(* Schneider Machine Expert - Basic project Tank_Level_Ultrasonic, file version 3.0.0.0 *)
(* ProjectInformations: Name=Tank_Level_Ultrasonic *)

HARDWARE
  Cpu 0: TM221CE16T
  ModuleExtensionObject 0: TM3AI4/G
  EthernetConfiguration: NetworkName=M221, IpAllocationMode=ByDhcp, IpAddress=192.168.1.10, SubnetMask=255.255.255.0
  SerialLineConfiguration: Baud=Baud19200, Parity=ParityEven, DataBits=DataBits8, StopBits=StopBits1, PhysicalMedium=PhysicalMediumRs485, TransmissionMode=TransmissionModeModbusRtu, SlaveId=1, Addressing=SlaveAddressing
  MastTask: UsePeriodScanMode=false, PeriodScan=100
  FastTask: Period=255
  CpuBehavior: StartingMode=StartAsPreviousState, AutoSaveRamOnEeprom=true, WatchdogPeriod=250

SYMBOLS  (address, symbol, comment, settings)
  %M0       PUMP_RUN  "Pump Running State"
  %M1       LEVEL_LOW  "Level below 1000mm - Start pump"
  %M2       LEVEL_HIGH  "Level above 1500mm - Stop pump"
  %M3       AUTO_CMD  "Auto mode pump command (hysteresis)"
  %M4       SENSOR_VALID  "Sensor reading valid (above dead band)"
  %M5       SENSOR_FAULT  "Sensor fault (below dead band)"
  %S0       SB_COLDSTART  "Indicates or executes a cold start (data initialized to default values)"
  %S1       SB_WARMSTART  "Indicates there was a warm start with data backup"
  %MW0      LVL_RAW  "Raw analog input value (0-10000)"
  %MW1      LVL_DISTANCE  "Distance from sensor in mm (300-5000)"
  %MW2      LVL_ACTUAL  "Actual tank level in mm (0-2000) for HMI"
  %MW10     SP_LOW  "Low level setpoint (1000mm)"
  %MW11     SP_HIGH  "High level setpoint (1500mm)"
  %I0.0     PB_START
  %I0.1     PB_STOP
  %I0.2     ESTOP
  %I0.3     SS_AUTO
  %Q0.0     PUMP_OUT
  %Q0.1     LT_RUN
  %Q0.2     LT_AUTO
  %Q0.3     LT_LOW
  %Q0.4     LT_HIGH
  %IW1.0    LVL_AIN  [Type=Type_4_20mA, Scope=Scope_Customized, Minimum=0, Maximum=10000]

POU Tank_Level_Ultrasonic
  (* SectionNumber=1 *)

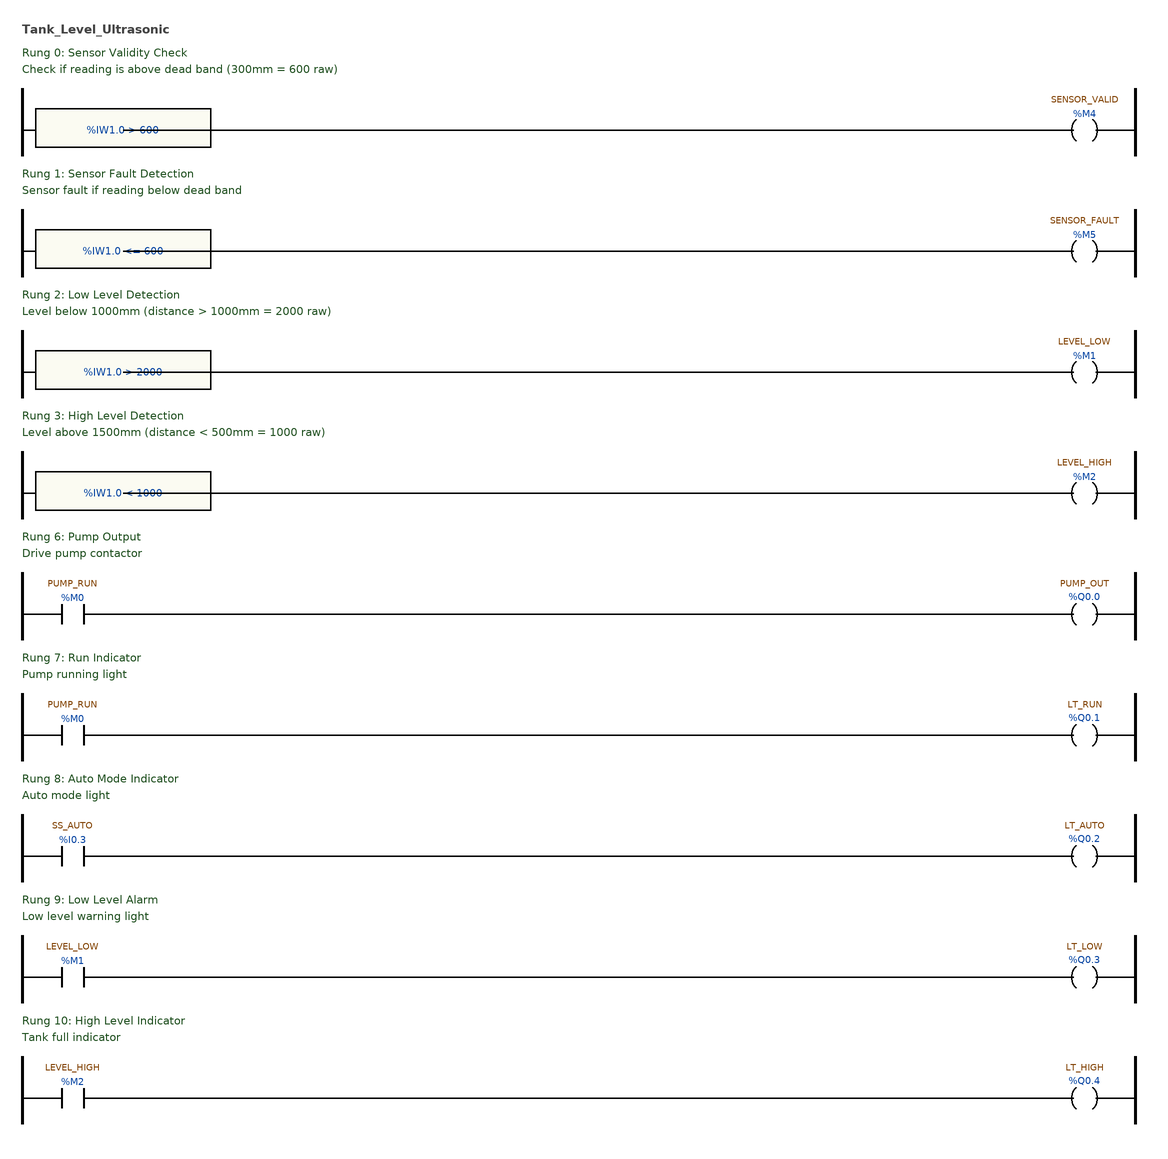

// Rung 0: Sensor Validity Check
// Check if reading is above dead band (300mm = 600 raw)
  LD [ %IW1.0 > 600 ]     (* LVL_AIN *)
  ST %M4                  (* SENSOR_VALID *)
  // as ST:
  //   SENSOR_VALID := LVL_AIN > 600;

// Rung 1: Sensor Fault Detection
// Sensor fault if reading below dead band
  LD [ %IW1.0 <= 600 ]    (* LVL_AIN *)
  ST %M5                  (* SENSOR_FAULT *)
  // as ST:
  //   SENSOR_FAULT := LVL_AIN <= 600;

// Rung 2: Low Level Detection
// Level below 1000mm (distance > 1000mm = 2000 raw)
  LD [ %IW1.0 > 2000 ]    (* LVL_AIN *)
  ST %M1                  (* LEVEL_LOW *)
  // as ST:
  //   LEVEL_LOW := LVL_AIN > 2000;

// Rung 3: High Level Detection
// Level above 1500mm (distance < 500mm = 1000 raw)
  LD [ %IW1.0 < 1000 ]    (* LVL_AIN *)
  ST %M2                  (* LEVEL_HIGH *)
  // as ST:
  //   LEVEL_HIGH := LVL_AIN < 1000;

// Rung 4: Auto Mode Hysteresis
// Start pump at low level, stop at high level (hysteresis 1000-1500mm)
  LD %M1                  (* LEVEL_LOW *)
  OR %M3                  (* AUTO_CMD *)
  ANDN %M2                (* LEVEL_HIGH *)
  AND %M4                 (* SENSOR_VALID *)
  ST %M3                  (* AUTO_CMD *)
  // as ST:
  //   AUTO_CMD := (LEVEL_LOW OR AUTO_CMD) AND NOT LEVEL_HIGH AND SENSOR_VALID;
  (* the ladder stored for this rung does not match its IL; not drawn *)

// Rung 5: Pump Run Control
// Pump runs in Auto mode with AUTO_CMD, or Manual with PB_START
  LD %I0.3                (* SS_AUTO *)
  AND %M3                 (* AUTO_CMD *)
  OR( %I0.0               (* PB_START *)
  OR %M0                  (* PUMP_RUN *)
  ANDN %I0.3              (* SS_AUTO *)
  )
  ANDN %I0.1              (* PB_STOP *)
  ANDN %I0.2              (* ESTOP *)
  AND %M4                 (* SENSOR_VALID *)
  ST %M0                  (* PUMP_RUN *)
  // as ST:
  //   PUMP_RUN := (SS_AUTO AND AUTO_CMD OR (PB_START OR PUMP_RUN) AND NOT SS_AUTO) AND NOT PB_STOP AND NOT ESTOP AND SENSOR_VALID;
  (* the ladder stored for this rung does not match its IL; not drawn *)

// Rung 6: Pump Output
// Drive pump contactor
  LD %M0                  (* PUMP_RUN *)
  ST %Q0.0                (* PUMP_OUT *)
  // as ST:
  //   PUMP_OUT := PUMP_RUN;

// Rung 7: Run Indicator
// Pump running light
  LD %M0                  (* PUMP_RUN *)
  ST %Q0.1                (* LT_RUN *)
  // as ST:
  //   LT_RUN := PUMP_RUN;

// Rung 8: Auto Mode Indicator
// Auto mode light
  LD %I0.3                (* SS_AUTO *)
  ST %Q0.2                (* LT_AUTO *)
  // as ST:
  //   LT_AUTO := SS_AUTO;

// Rung 9: Low Level Alarm
// Low level warning light
  LD %M1                  (* LEVEL_LOW *)
  ST %Q0.3                (* LT_LOW *)
  // as ST:
  //   LT_LOW := LEVEL_LOW;

// Rung 10: High Level Indicator
// Tank full indicator
  LD %M2                  (* LEVEL_HIGH *)
  ST %Q0.4                (* LT_HIGH *)
  // as ST:
  //   LT_HIGH := LEVEL_HIGH;

// Rung 11: HMI Raw Level
// Copy raw analog value to %MW0 for HMI access
  LD %S1                  (* SB_WARMSTART *)
  OR %S0                  (* SB_COLDSTART *)
  [%MW0 := %IW1.0]        (* LVL_RAW, LVL_AIN *)
  // as ST:
  //   IF SB_WARMSTART OR SB_COLDSTART THEN LVL_RAW := LVL_AIN; END_IF;
  (* the ladder stored for this rung does not match its IL; not drawn *)

// Rung 12: HMI Actual Level
// Calculate actual tank level: 2000 - (distance). Scale: raw/2 = distance(mm), level = 2000 - distance
  LD %S1                  (* SB_WARMSTART *)
  OR %S0                  (* SB_COLDSTART *)
  [%MW1 := %MW0 * 5000 / 10000](* LVL_DISTANCE, LVL_RAW *)
  [%MW2 := 2000 - %MW1]   (* LVL_ACTUAL, LVL_DISTANCE *)
  // as ST:
  //   IF SB_WARMSTART OR SB_COLDSTART THEN LVL_DISTANCE := LVL_RAW * 5000 / 10000; END_IF;
  //   IF SB_WARMSTART OR SB_COLDSTART THEN LVL_ACTUAL := 2000 - LVL_DISTANCE; END_IF;
  (* the ladder stored for this rung does not match its IL; not drawn *)
